INTERFACE I_LimitedStringBuilder

METHOD  Append : I_StringBuilder // Append text to t current build string.
VAR_INPUT
	Text : STRING; //Text to append to current build string
END_VAR
END_METHOD

METHOD Left : I_StringBuilder
VAR_INPUT
	Count : INT;
END_VAR
END_METHOD

PROPERTY Length : INT
GET
END_GET
END_PROPERTY

METHOD Reset : I_LimitedStringBuilder //Reset current build string to an empty string.
END_METHOD

METHOD Right : I_StringBuilder
VAR_INPUT
	Count : INT;
END_VAR
END_METHOD

METHOD ToString : STRING //Returns current build string.
END_METHOD

END_INTERFACE

(* stored: Version 1.1.0.1, ProductVersion 3.1.4024.12
   Itf I_LimitedStringBuilder: Id {194bb722-4e19-4a72-9bf7-057dc58bb68e}
   Method Append: Id {c1fd36d6-9aa3-4352-9719-226e4a16c216}
   Method Left: Id {2f9c4273-e955-4025-93f9-c4ff974a7b9f}
   Property Length: Id {6672f6f6-8923-436c-8365-e1ec6007f746}
   Get Get: Id {894ce71b-c68f-48e0-8db7-33d19b2c0a3f}
   Method Reset: Id {0267de3b-ea97-4e81-b5fa-899dfdee3f2c}
   Method Right: Id {e124d91a-18be-4ab9-8ee1-853b8fad81b2}
   Method ToString: Id {9510ec58-ffae-406c-b1a3-226f94c7f534} *)
